PROGRAM P_Simulator
VAR
	fbCylinderSim : FB_CylinderSimulator;
END_VAR
VAR_INPUT
	stSimSystemOutputs : ST_inputs_analog;
	eCraneState : E_CraneStatus;
	stSimInputs : ST_ValvePos;
END_VAR

IF eCraneState <> E_CraneStatus.Off THEN // <> = !=
	fbCylinderSim(ssMethodType := 1,
		fNormalizedValveInput := stSimInputs.rCylinderValve,
		fPistonPosition_m => stSimSystemOutputs.fPistonPos,
		fPistonSidePressure_bar => stSimSystemOutputs.fP_piston,
		fRodSidePressure_bar => stSimSystemOutputs.fP_rod);
ELSE
	fbCylinderSim(ssMethodType := 0);
END_IF

END_PROGRAM

(* stored: Version 1.1.0.1
   POU P_Simulator: Id {842435b2-f633-4562-a126-ecf8133e2003}, SpecialFunc None *)
